{attribute 'qualified_only'}
VAR_GLOBAL
	Inputs  AT %I* : ST_Bridge_TSCS;	// Inputs
	Outputs AT %Q* : ST_Bridge_TDU;		// Outputs
END_VAR

(* stored: Version 1.1.0.1, ProductVersion 3.1.4024.3
   GVL BridgeTerminal_TSCS: Id {446546ba-e92c-4390-aff6-c7d51684de6a} *)
